{attribute 'qualified_only'}
VAR_GLOBAL
    {attribute 'pytmc' := 'pv: DREAM:MC:MMS:Y '}
    {attribute 'TcLinkTo' := '.bLimitForwardEnable  := TIIB[DRL_05_EL7047_E1]^STM Status^Status^Digital input 1;
                              .bLimitBackwardEnable := TIIB[DRL_05_EL7047_E1]^STM Status^Status^Digital input 2;
                              .nRawEncoderULINT     := TIIB[DRL_05_EL5042_E2]^FB Inputs Channel 1^Position'}
    M1: DUT_MotionStage := (sName := 'DREAM:MC:MMS:Y ');

    {attribute 'pytmc' := 'pv: DREAM:COIL:MMS:ROLL '}
    {attribute 'TcLinkTo' := '.bLimitForwardEnable  := TIIB[DRL_05_EL7047_E3]^STM Status^Status^Digital input 1;
                              .bLimitBackwardEnable := TIIB[DRL_05_EL7047_E3]^STM Status^Status^Digital input 2;
                              .nRawEncoderULINT     := TIIB[DRL_05_EL5042_E2]^FB Inputs Channel 2^Position'}
    M2: DUT_MotionStage := (sName := 'DREAM:COIL:MMS:ROLL ');

    {attribute 'pytmc' := 'pv: DREAM:COIL:MMS:YAW '}
    {attribute 'TcLinkTo' := '.bLimitForwardEnable  := TIIB[DRL_05_EL7047_E4]^STM Status^Status^Digital input 1;
                              .bLimitBackwardEnable := TIIB[DRL_05_EL7047_E4]^STM Status^Status^Digital input 2;
                              .nRawEncoderULINT     := TIIB[DRL_05_EL5042_E5]^FB Inputs Channel 1^Position'}
    M3: DUT_MotionStage := (sName := 'DREAM:COIL:MMS:YAW ');

    {attribute 'pytmc' := 'pv: DREAM:GSJP:MMS:X '}
    {attribute 'TcLinkTo' := '.bLimitForwardEnable  := TIIB[DRL_05_EL7047_E6]^STM Status^Status^Digital input 1;
                              .bLimitBackwardEnable := TIIB[DRL_05_EL7047_E6]^STM Status^Status^Digital input 2;
                              .nRawEncoderULINT     := TIIB[DRL_05_EL5042_E5]^FB Inputs Channel 2^Position'}
    M4: DUT_MotionStage := (sName := 'DREAM:GSJP:MMS:X ');

    {attribute 'pytmc' := 'pv: DREAM:GSJP:MMS:Z '}
    {attribute 'TcLinkTo' := '.bLimitForwardEnable  := TIIB[DRL_05_EL7047_E7]^STM Status^Status^Digital input 2;
                              .bLimitBackwardEnable := TIIB[DRL_05_EL7047_E7]^STM Status^Status^Digital input 1;
                              .nRawEncoderULINT     := TIIB[DRL_05_EL5042_E8]^FB Inputs Channel 1^Position'}
    M5: DUT_MotionStage := (sName := 'DREAM:GSJP:MMS:Z ');

    {attribute 'pytmc' := 'pv: DREAM:GSJN:MMS:X'}
    {attribute 'TcLinkTo' := '.bLimitForwardEnable  := TIIB[DRL_05_EL7047_E9]^STM Status^Status^Digital input 2;
                              .bLimitBackwardEnable := TIIB[DRL_05_EL7047_E9]^STM Status^Status^Digital input 1;
                              .nRawEncoderULINT     := TIIB[DRL_05_EL5042_E8]^FB Inputs Channel 2^Position'}
    M6: DUT_MotionStage := (sName := 'DREAM:GSJN:MMS:X');

    {attribute 'pytmc' := 'pv: DREAM:GSJN:MMS:Y'}
    {attribute 'TcLinkTo' := '.bLimitForwardEnable  := TIIB[DRL_05_EL7047_E10]^STM Status^Status^Digital input 2;
                              .bLimitBackwardEnable := TIIB[DRL_05_EL7047_E10]^STM Status^Status^Digital input 1;
                              .nRawEncoderULINT     := TIIB[DRL_05_EL5042_E11]^FB Inputs Channel 1^Position'}
    M7: DUT_MotionStage := (sName := 'DREAM:GSJN:MMS:Y');

    {attribute 'pytmc' := 'pv: DREAM:GSJN:MMS:Z'}
    {attribute 'TcLinkTo' := '.bLimitForwardEnable  := TIIB[DRL_05_EL7047_E12]^STM Status^Status^Digital input 1;
                              .bLimitBackwardEnable := TIIB[DRL_05_EL7047_E12]^STM Status^Status^Digital input 2;
                              .nRawEncoderULINT     := TIIB[DRL_05_EL5042_E11]^FB Inputs Channel 2^Position'}
    M8: DUT_MotionStage := (sName := 'DREAM:GSJN:MMS:Z');


END_VAR

(* stored: Version 1.1.0.1, ProductVersion 3.1.4024.12
   GVL Main: Id {18d82037-8457-400f-b1ad-ea349db133b4} *)
